// TIA Portal V19 export
FUNCTION "SUBOUTPUT" : Void   // FC4, LAD
{ S7_Optimized_Access := 'TRUE' }
// stored: SetENOAutomatically false
BEGIN

REGION Network 1: HOOTER
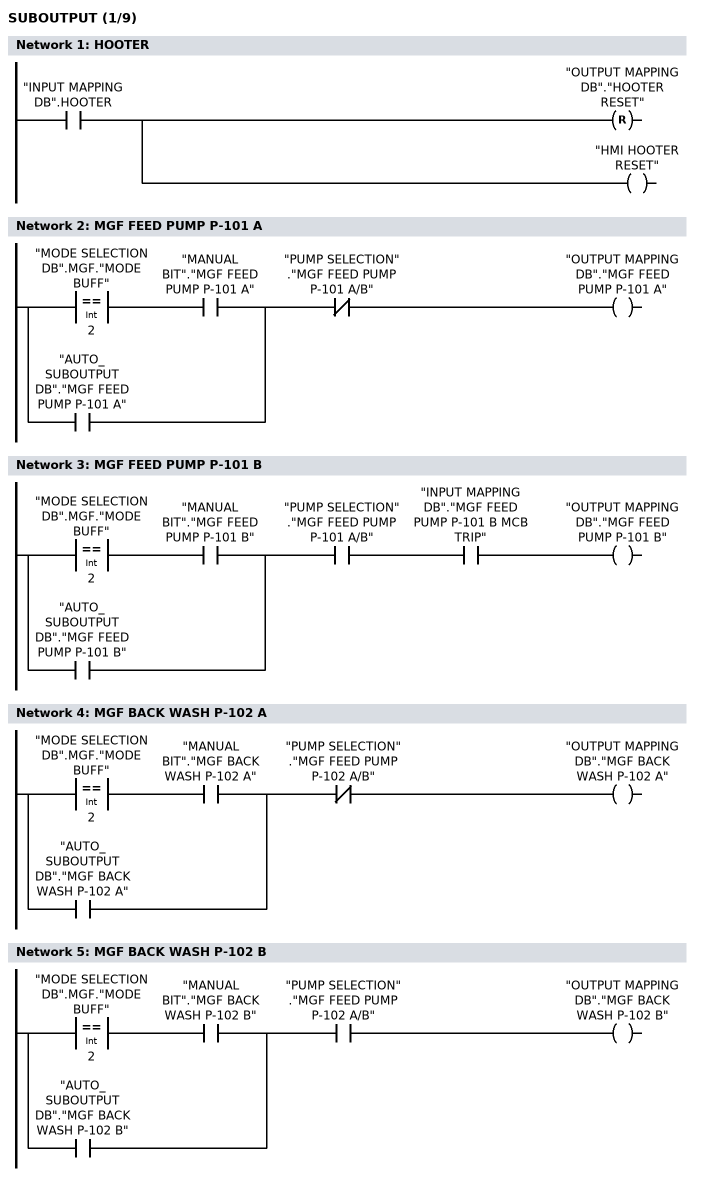
   RUNG wire#powerrail
      Contact( "INPUT MAPPING DB".HOOTER )
      wire#w1
      R_Coil( "OUTPUT MAPPING DB"."HOOTER RESET" )
   END_RUNG
   RUNG wire#w1
      Coil( "HMI HOOTER RESET" )
   END_RUNG
   // the same network as SCL:
   IF "INPUT MAPPING DB".HOOTER THEN "OUTPUT MAPPING DB"."HOOTER RESET" := FALSE; END_IF;
   "HMI HOOTER RESET" := "INPUT MAPPING DB".HOOTER;
END_REGION

REGION Network 2: MGF FEED PUMP P-101 A
   RUNG wire#powerrail
      { S7_Templates := "SrcType := Int" } EQ_Contact(in1 := "MODE SELECTION DB".MGF."MODE BUFF", in2 := 2)
      Contact( "MANUAL BIT"."MGF FEED PUMP P-101 A" )
      wire#w1
      I_Contact( "PUMP SELECTION"."MGF FEED PUMP P-101 A/B" )
      Coil( "OUTPUT MAPPING DB"."MGF FEED PUMP P-101 A" )
   END_RUNG
   RUNG wire#powerrail
      Contact( "AUTO_SUBOUTPUT DB"."MGF FEED PUMP P-101 A" )
   END_RUNG wire#w1
   // the same network as SCL:
   "OUTPUT MAPPING DB"."MGF FEED PUMP P-101 A" := ((("MODE SELECTION DB".MGF."MODE BUFF" = 2) AND "MANUAL BIT"."MGF FEED PUMP P-101 A") OR "AUTO_SUBOUTPUT DB"."MGF FEED PUMP P-101 A") AND NOT "PUMP SELECTION"."MGF FEED PUMP P-101 A/B";
END_REGION

REGION Network 3: MGF FEED PUMP P-101 B
   RUNG wire#powerrail
      { S7_Templates := "SrcType := Int" } EQ_Contact(in1 := "MODE SELECTION DB".MGF."MODE BUFF", in2 := 2)
      Contact( "MANUAL BIT"."MGF FEED PUMP P-101 B" )
      wire#w1
      Contact( "PUMP SELECTION"."MGF FEED PUMP P-101 A/B" )
      Contact( "INPUT MAPPING DB"."MGF FEED PUMP P-101 B MCB TRIP" )
      Coil( "OUTPUT MAPPING DB"."MGF FEED PUMP P-101 B" )
   END_RUNG
   RUNG wire#powerrail
      Contact( "AUTO_SUBOUTPUT DB"."MGF FEED PUMP P-101 B" )
   END_RUNG wire#w1
   // the same network as SCL:
   "OUTPUT MAPPING DB"."MGF FEED PUMP P-101 B" := ((("MODE SELECTION DB".MGF."MODE BUFF" = 2) AND "MANUAL BIT"."MGF FEED PUMP P-101 B") OR "AUTO_SUBOUTPUT DB"."MGF FEED PUMP P-101 B") AND "PUMP SELECTION"."MGF FEED PUMP P-101 A/B" AND "INPUT MAPPING DB"."MGF FEED PUMP P-101 B MCB TRIP";
END_REGION

REGION Network 4: MGF BACK WASH P-102 A
   RUNG wire#powerrail
      { S7_Templates := "SrcType := Int" } EQ_Contact(in1 := "MODE SELECTION DB".MGF."MODE BUFF", in2 := 2)
      Contact( "MANUAL BIT"."MGF BACK WASH P-102 A" )
      wire#w1
      I_Contact( "PUMP SELECTION"."MGF FEED PUMP P-102 A/B" )
      Coil( "OUTPUT MAPPING DB"."MGF BACK WASH P-102 A" )
   END_RUNG
   RUNG wire#powerrail
      Contact( "AUTO_SUBOUTPUT DB"."MGF BACK WASH P-102 A" )
   END_RUNG wire#w1
   // the same network as SCL:
   "OUTPUT MAPPING DB"."MGF BACK WASH P-102 A" := ((("MODE SELECTION DB".MGF."MODE BUFF" = 2) AND "MANUAL BIT"."MGF BACK WASH P-102 A") OR "AUTO_SUBOUTPUT DB"."MGF BACK WASH P-102 A") AND NOT "PUMP SELECTION"."MGF FEED PUMP P-102 A/B";
END_REGION

REGION Network 5: MGF BACK WASH P-102 B
   RUNG wire#powerrail
      { S7_Templates := "SrcType := Int" } EQ_Contact(in1 := "MODE SELECTION DB".MGF."MODE BUFF", in2 := 2)
      Contact( "MANUAL BIT"."MGF BACK WASH P-102 B" )
      wire#w1
      Contact( "PUMP SELECTION"."MGF FEED PUMP P-102 A/B" )
      Coil( "OUTPUT MAPPING DB"."MGF BACK WASH P-102 B" )
   END_RUNG
   RUNG wire#powerrail
      Contact( "AUTO_SUBOUTPUT DB"."MGF BACK WASH P-102 B" )
   END_RUNG wire#w1
   // the same network as SCL:
   "OUTPUT MAPPING DB"."MGF BACK WASH P-102 B" := ((("MODE SELECTION DB".MGF."MODE BUFF" = 2) AND "MANUAL BIT"."MGF BACK WASH P-102 B") OR "AUTO_SUBOUTPUT DB"."MGF BACK WASH P-102 B") AND "PUMP SELECTION"."MGF FEED PUMP P-102 A/B";
END_REGION

REGION Network 6: UF FEED PUMP P-103 A
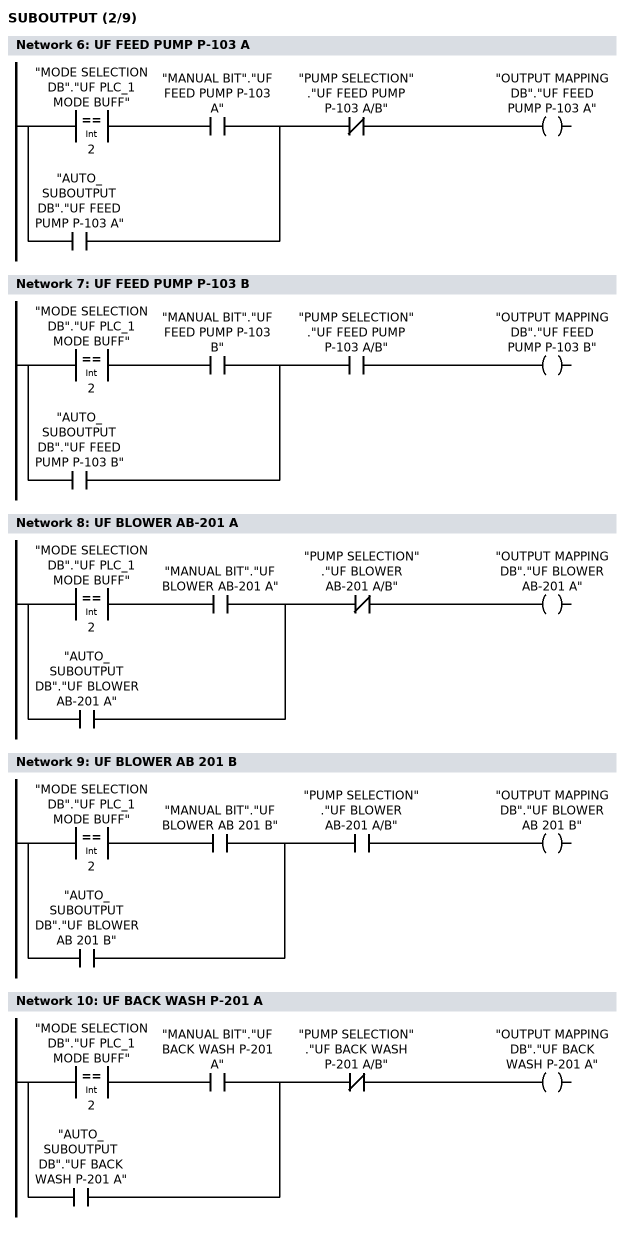
   RUNG wire#powerrail
      { S7_Templates := "SrcType := Int" } EQ_Contact(in1 := "MODE SELECTION DB"."UF PLC_1 MODE BUFF", in2 := 2)
      Contact( "MANUAL BIT"."UF FEED PUMP P-103 A" )
      wire#w1
      I_Contact( "PUMP SELECTION"."UF FEED PUMP P-103 A/B" )
      Coil( "OUTPUT MAPPING DB"."UF FEED PUMP P-103 A" )
   END_RUNG
   RUNG wire#powerrail
      Contact( "AUTO_SUBOUTPUT DB"."UF FEED PUMP P-103 A" )
   END_RUNG wire#w1
   // the same network as SCL:
   "OUTPUT MAPPING DB"."UF FEED PUMP P-103 A" := ((("MODE SELECTION DB"."UF PLC_1 MODE BUFF" = 2) AND "MANUAL BIT"."UF FEED PUMP P-103 A") OR "AUTO_SUBOUTPUT DB"."UF FEED PUMP P-103 A") AND NOT "PUMP SELECTION"."UF FEED PUMP P-103 A/B";
END_REGION

REGION Network 7: UF FEED PUMP P-103 B
   RUNG wire#powerrail
      { S7_Templates := "SrcType := Int" } EQ_Contact(in1 := "MODE SELECTION DB"."UF PLC_1 MODE BUFF", in2 := 2)
      Contact( "MANUAL BIT"."UF FEED PUMP P-103 B" )
      wire#w1
      Contact( "PUMP SELECTION"."UF FEED PUMP P-103 A/B" )
      Coil( "OUTPUT MAPPING DB"."UF FEED PUMP P-103 B" )
   END_RUNG
   RUNG wire#powerrail
      Contact( "AUTO_SUBOUTPUT DB"."UF FEED PUMP P-103 B" )
   END_RUNG wire#w1
   // the same network as SCL:
   "OUTPUT MAPPING DB"."UF FEED PUMP P-103 B" := ((("MODE SELECTION DB"."UF PLC_1 MODE BUFF" = 2) AND "MANUAL BIT"."UF FEED PUMP P-103 B") OR "AUTO_SUBOUTPUT DB"."UF FEED PUMP P-103 B") AND "PUMP SELECTION"."UF FEED PUMP P-103 A/B";
END_REGION

REGION Network 8: UF BLOWER AB-201 A
   RUNG wire#powerrail
      { S7_Templates := "SrcType := Int" } EQ_Contact(in1 := "MODE SELECTION DB"."UF PLC_1 MODE BUFF", in2 := 2)
      Contact( "MANUAL BIT"."UF BLOWER AB-201 A" )
      wire#w1
      I_Contact( "PUMP SELECTION"."UF BLOWER AB-201 A/B" )
      Coil( "OUTPUT MAPPING DB"."UF BLOWER AB-201 A" )
   END_RUNG
   RUNG wire#powerrail
      Contact( "AUTO_SUBOUTPUT DB"."UF BLOWER AB-201 A" )
   END_RUNG wire#w1
   // the same network as SCL:
   "OUTPUT MAPPING DB"."UF BLOWER AB-201 A" := ((("MODE SELECTION DB"."UF PLC_1 MODE BUFF" = 2) AND "MANUAL BIT"."UF BLOWER AB-201 A") OR "AUTO_SUBOUTPUT DB"."UF BLOWER AB-201 A") AND NOT "PUMP SELECTION"."UF BLOWER AB-201 A/B";
END_REGION

REGION Network 9: UF BLOWER AB 201 B
   RUNG wire#powerrail
      { S7_Templates := "SrcType := Int" } EQ_Contact(in1 := "MODE SELECTION DB"."UF PLC_1 MODE BUFF", in2 := 2)
      Contact( "MANUAL BIT"."UF BLOWER AB 201 B" )
      wire#w1
      Contact( "PUMP SELECTION"."UF BLOWER AB-201 A/B" )
      Coil( "OUTPUT MAPPING DB"."UF BLOWER AB 201 B" )
   END_RUNG
   RUNG wire#powerrail
      Contact( "AUTO_SUBOUTPUT DB"."UF BLOWER AB 201 B" )
   END_RUNG wire#w1
   // the same network as SCL:
   "OUTPUT MAPPING DB"."UF BLOWER AB 201 B" := ((("MODE SELECTION DB"."UF PLC_1 MODE BUFF" = 2) AND "MANUAL BIT"."UF BLOWER AB 201 B") OR "AUTO_SUBOUTPUT DB"."UF BLOWER AB 201 B") AND "PUMP SELECTION"."UF BLOWER AB-201 A/B";
END_REGION

REGION Network 10: UF BACK WASH P-201 A
   RUNG wire#powerrail
      { S7_Templates := "SrcType := Int" } EQ_Contact(in1 := "MODE SELECTION DB"."UF PLC_1 MODE BUFF", in2 := 2)
      Contact( "MANUAL BIT"."UF BACK WASH P-201 A" )
      wire#w1
      I_Contact( "PUMP SELECTION"."UF BACK WASH P-201 A/B" )
      Coil( "OUTPUT MAPPING DB"."UF BACK WASH P-201 A" )
   END_RUNG
   RUNG wire#powerrail
      Contact( "AUTO_SUBOUTPUT DB"."UF BACK WASH P-201 A" )
   END_RUNG wire#w1
   // the same network as SCL:
   "OUTPUT MAPPING DB"."UF BACK WASH P-201 A" := ((("MODE SELECTION DB"."UF PLC_1 MODE BUFF" = 2) AND "MANUAL BIT"."UF BACK WASH P-201 A") OR "AUTO_SUBOUTPUT DB"."UF BACK WASH P-201 A") AND NOT "PUMP SELECTION"."UF BACK WASH P-201 A/B";
END_REGION

REGION Network 11: UF BACK WASH P-201 B
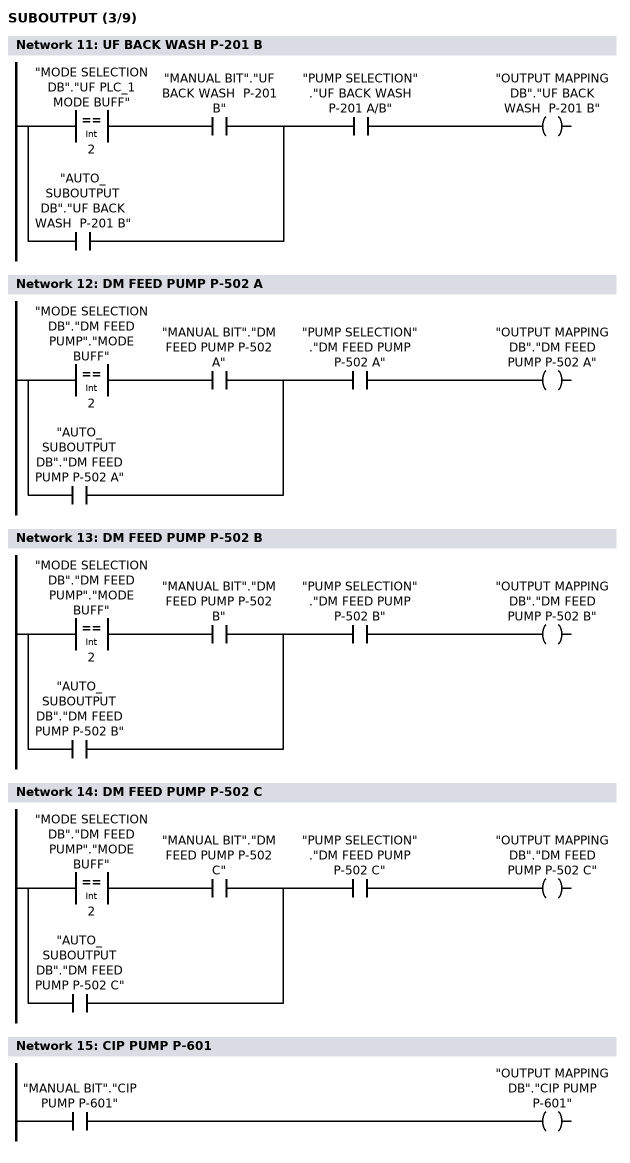
   RUNG wire#powerrail
      { S7_Templates := "SrcType := Int" } EQ_Contact(in1 := "MODE SELECTION DB"."UF PLC_1 MODE BUFF", in2 := 2)
      Contact( "MANUAL BIT"."UF BACK WASH  P-201 B" )
      wire#w1
      Contact( "PUMP SELECTION"."UF BACK WASH P-201 A/B" )
      Coil( "OUTPUT MAPPING DB"."UF BACK WASH  P-201 B" )
   END_RUNG
   RUNG wire#powerrail
      Contact( "AUTO_SUBOUTPUT DB"."UF BACK WASH  P-201 B" )
   END_RUNG wire#w1
   // the same network as SCL:
   "OUTPUT MAPPING DB"."UF BACK WASH  P-201 B" := ((("MODE SELECTION DB"."UF PLC_1 MODE BUFF" = 2) AND "MANUAL BIT"."UF BACK WASH  P-201 B") OR "AUTO_SUBOUTPUT DB"."UF BACK WASH  P-201 B") AND "PUMP SELECTION"."UF BACK WASH P-201 A/B";
END_REGION

REGION Network 12: DM FEED PUMP P-502 A
   RUNG wire#powerrail
      { S7_Templates := "SrcType := Int" } EQ_Contact(in1 := "MODE SELECTION DB"."DM FEED PUMP"."MODE BUFF", in2 := 2)
      Contact( "MANUAL BIT"."DM FEED PUMP P-502 A" )
      wire#w1
      Contact( "PUMP SELECTION"."DM FEED PUMP P-502 A" )
      Coil( "OUTPUT MAPPING DB"."DM FEED PUMP P-502 A" )
   END_RUNG
   RUNG wire#powerrail
      Contact( "AUTO_SUBOUTPUT DB"."DM FEED PUMP P-502 A" )
   END_RUNG wire#w1
   // the same network as SCL:
   "OUTPUT MAPPING DB"."DM FEED PUMP P-502 A" := ((("MODE SELECTION DB"."DM FEED PUMP"."MODE BUFF" = 2) AND "MANUAL BIT"."DM FEED PUMP P-502 A") OR "AUTO_SUBOUTPUT DB"."DM FEED PUMP P-502 A") AND "PUMP SELECTION"."DM FEED PUMP P-502 A";
END_REGION

REGION Network 13: DM FEED PUMP P-502 B
   RUNG wire#powerrail
      { S7_Templates := "SrcType := Int" } EQ_Contact(in1 := "MODE SELECTION DB"."DM FEED PUMP"."MODE BUFF", in2 := 2)
      Contact( "MANUAL BIT"."DM FEED PUMP P-502 B" )
      wire#w1
      Contact( "PUMP SELECTION"."DM FEED PUMP P-502 B" )
      Coil( "OUTPUT MAPPING DB"."DM FEED PUMP P-502 B" )
   END_RUNG
   RUNG wire#powerrail
      Contact( "AUTO_SUBOUTPUT DB"."DM FEED PUMP P-502 B" )
   END_RUNG wire#w1
   // the same network as SCL:
   "OUTPUT MAPPING DB"."DM FEED PUMP P-502 B" := ((("MODE SELECTION DB"."DM FEED PUMP"."MODE BUFF" = 2) AND "MANUAL BIT"."DM FEED PUMP P-502 B") OR "AUTO_SUBOUTPUT DB"."DM FEED PUMP P-502 B") AND "PUMP SELECTION"."DM FEED PUMP P-502 B";
END_REGION

REGION Network 14: DM FEED PUMP P-502 C
   RUNG wire#powerrail
      { S7_Templates := "SrcType := Int" } EQ_Contact(in1 := "MODE SELECTION DB"."DM FEED PUMP"."MODE BUFF", in2 := 2)
      Contact( "MANUAL BIT"."DM FEED PUMP P-502 C" )
      wire#w1
      Contact( "PUMP SELECTION"."DM FEED PUMP P-502 C" )
      Coil( "OUTPUT MAPPING DB"."DM FEED PUMP P-502 C" )
   END_RUNG
   RUNG wire#powerrail
      Contact( "AUTO_SUBOUTPUT DB"."DM FEED PUMP P-502 C" )
   END_RUNG wire#w1
   // the same network as SCL:
   "OUTPUT MAPPING DB"."DM FEED PUMP P-502 C" := ((("MODE SELECTION DB"."DM FEED PUMP"."MODE BUFF" = 2) AND "MANUAL BIT"."DM FEED PUMP P-502 C") OR "AUTO_SUBOUTPUT DB"."DM FEED PUMP P-502 C") AND "PUMP SELECTION"."DM FEED PUMP P-502 C";
END_REGION

REGION Network 15: CIP PUMP P-601
   RUNG wire#powerrail
      Contact( "MANUAL BIT"."CIP PUMP P-601" )
      Coil( "OUTPUT MAPPING DB"."CIP PUMP P-601" )
   END_RUNG
   // the same network as SCL:
   "OUTPUT MAPPING DB"."CIP PUMP P-601" := "MANUAL BIT"."CIP PUMP P-601";
END_REGION

REGION Network 16: BACK WASH RECOVERY P-801 A
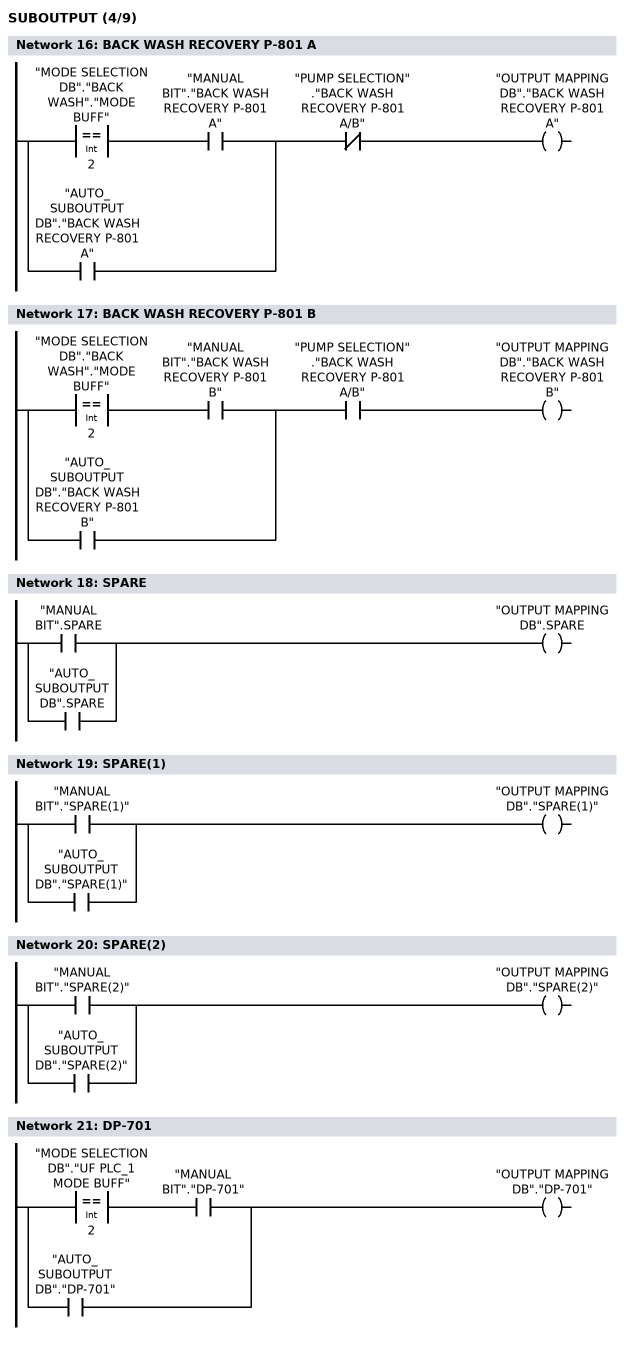
   RUNG wire#powerrail
      { S7_Templates := "SrcType := Int" } EQ_Contact(in1 := "MODE SELECTION DB"."BACK WASH"."MODE BUFF", in2 := 2)
      Contact( "MANUAL BIT"."BACK WASH RECOVERY P-801 A" )
      wire#w1
      I_Contact( "PUMP SELECTION"."BACK WASH RECOVERY P-801 A/B" )
      Coil( "OUTPUT MAPPING DB"."BACK WASH RECOVERY P-801 A" )
   END_RUNG
   RUNG wire#powerrail
      Contact( "AUTO_SUBOUTPUT DB"."BACK WASH RECOVERY P-801 A" )
   END_RUNG wire#w1
   // the same network as SCL:
   "OUTPUT MAPPING DB"."BACK WASH RECOVERY P-801 A" := ((("MODE SELECTION DB"."BACK WASH"."MODE BUFF" = 2) AND "MANUAL BIT"."BACK WASH RECOVERY P-801 A") OR "AUTO_SUBOUTPUT DB"."BACK WASH RECOVERY P-801 A") AND NOT "PUMP SELECTION"."BACK WASH RECOVERY P-801 A/B";
END_REGION

REGION Network 17: BACK WASH RECOVERY P-801 B
   RUNG wire#powerrail
      { S7_Templates := "SrcType := Int" } EQ_Contact(in1 := "MODE SELECTION DB"."BACK WASH"."MODE BUFF", in2 := 2)
      Contact( "MANUAL BIT"."BACK WASH RECOVERY P-801 B" )
      wire#w1
      Contact( "PUMP SELECTION"."BACK WASH RECOVERY P-801 A/B" )
      Coil( "OUTPUT MAPPING DB"."BACK WASH RECOVERY P-801 B" )
   END_RUNG
   RUNG wire#powerrail
      Contact( "AUTO_SUBOUTPUT DB"."BACK WASH RECOVERY P-801 B" )
   END_RUNG wire#w1
   // the same network as SCL:
   "OUTPUT MAPPING DB"."BACK WASH RECOVERY P-801 B" := ((("MODE SELECTION DB"."BACK WASH"."MODE BUFF" = 2) AND "MANUAL BIT"."BACK WASH RECOVERY P-801 B") OR "AUTO_SUBOUTPUT DB"."BACK WASH RECOVERY P-801 B") AND "PUMP SELECTION"."BACK WASH RECOVERY P-801 A/B";
END_REGION

REGION Network 18: SPARE
   RUNG wire#powerrail
      Contact( "MANUAL BIT".SPARE )
      wire#w1
      Coil( "OUTPUT MAPPING DB".SPARE )
   END_RUNG
   RUNG wire#powerrail
      Contact( "AUTO_SUBOUTPUT DB".SPARE )
   END_RUNG wire#w1
   // the same network as SCL:
   "OUTPUT MAPPING DB".SPARE := "MANUAL BIT".SPARE OR "AUTO_SUBOUTPUT DB".SPARE;
END_REGION

REGION Network 19: SPARE(1)
   RUNG wire#powerrail
      Contact( "MANUAL BIT"."SPARE(1)" )
      wire#w1
      Coil( "OUTPUT MAPPING DB"."SPARE(1)" )
   END_RUNG
   RUNG wire#powerrail
      Contact( "AUTO_SUBOUTPUT DB"."SPARE(1)" )
   END_RUNG wire#w1
   // the same network as SCL:
   "OUTPUT MAPPING DB"."SPARE(1)" := "MANUAL BIT"."SPARE(1)" OR "AUTO_SUBOUTPUT DB"."SPARE(1)";
END_REGION

REGION Network 20: SPARE(2)
   RUNG wire#powerrail
      Contact( "MANUAL BIT"."SPARE(2)" )
      wire#w1
      Coil( "OUTPUT MAPPING DB"."SPARE(2)" )
   END_RUNG
   RUNG wire#powerrail
      Contact( "AUTO_SUBOUTPUT DB"."SPARE(2)" )
   END_RUNG wire#w1
   // the same network as SCL:
   "OUTPUT MAPPING DB"."SPARE(2)" := "MANUAL BIT"."SPARE(2)" OR "AUTO_SUBOUTPUT DB"."SPARE(2)";
END_REGION

REGION Network 21: DP-701
   RUNG wire#powerrail
      { S7_Templates := "SrcType := Int" } EQ_Contact(in1 := "MODE SELECTION DB"."UF PLC_1 MODE BUFF", in2 := 2)
      Contact( "MANUAL BIT"."DP-701" )
      wire#w1
      Coil( "OUTPUT MAPPING DB"."DP-701" )
   END_RUNG
   RUNG wire#powerrail
      Contact( "AUTO_SUBOUTPUT DB"."DP-701" )
   END_RUNG wire#w1
   // the same network as SCL:
   "OUTPUT MAPPING DB"."DP-701" := (("MODE SELECTION DB"."UF PLC_1 MODE BUFF" = 2) AND "MANUAL BIT"."DP-701") OR "AUTO_SUBOUTPUT DB"."DP-701";
END_REGION

REGION Network 22: DP-702
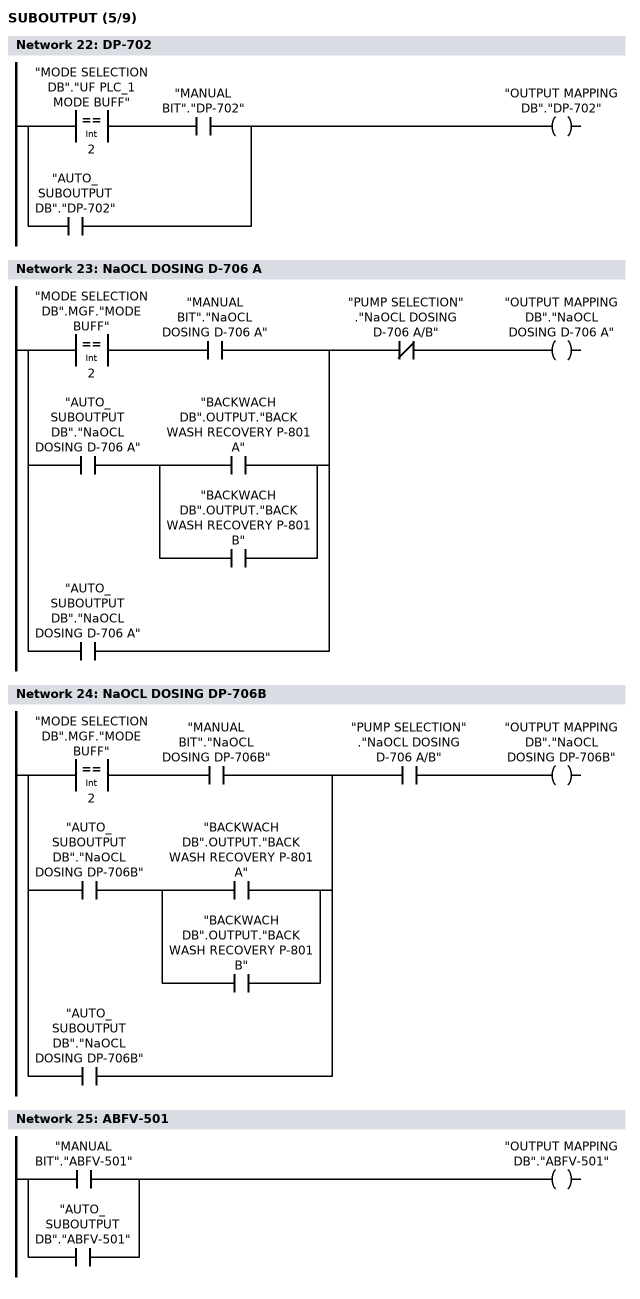
   RUNG wire#powerrail
      { S7_Templates := "SrcType := Int" } EQ_Contact(in1 := "MODE SELECTION DB"."UF PLC_1 MODE BUFF", in2 := 2)
      Contact( "MANUAL BIT"."DP-702" )
      wire#w1
      Coil( "OUTPUT MAPPING DB"."DP-702" )
   END_RUNG
   RUNG wire#powerrail
      Contact( "AUTO_SUBOUTPUT DB"."DP-702" )
   END_RUNG wire#w1
   // the same network as SCL:
   "OUTPUT MAPPING DB"."DP-702" := (("MODE SELECTION DB"."UF PLC_1 MODE BUFF" = 2) AND "MANUAL BIT"."DP-702") OR "AUTO_SUBOUTPUT DB"."DP-702";
END_REGION

REGION Network 23: NaOCL DOSING D-706 A
   RUNG wire#powerrail
      { S7_Templates := "SrcType := Int" } EQ_Contact(in1 := "MODE SELECTION DB".MGF."MODE BUFF", in2 := 2)
      Contact( "MANUAL BIT"."NaOCL DOSING D-706 A" )
      wire#w1
      I_Contact( "PUMP SELECTION"."NaOCL DOSING D-706 A/B" )
      Coil( "OUTPUT MAPPING DB"."NaOCL DOSING D-706 A" )
   END_RUNG
   RUNG wire#powerrail
      Contact( "AUTO_SUBOUTPUT DB"."NaOCL DOSING D-706 A" )
      wire#w2
      Contact( "BACKWACH DB".OUTPUT."BACK WASH RECOVERY P-801 A" )
   END_RUNG wire#w1
   RUNG wire#w2
      Contact( "BACKWACH DB".OUTPUT."BACK WASH RECOVERY P-801 B" )
   END_RUNG wire#w1
   RUNG wire#powerrail
      Contact( "AUTO_SUBOUTPUT DB"."NaOCL DOSING D-706 A" )
   END_RUNG wire#w1
   // the same network as SCL:
   "OUTPUT MAPPING DB"."NaOCL DOSING D-706 A" := ((("MODE SELECTION DB".MGF."MODE BUFF" = 2) AND "MANUAL BIT"."NaOCL DOSING D-706 A") OR ("AUTO_SUBOUTPUT DB"."NaOCL DOSING D-706 A" AND ("BACKWACH DB".OUTPUT."BACK WASH RECOVERY P-801 A" OR "BACKWACH DB".OUTPUT."BACK WASH RECOVERY P-801 B")) OR "AUTO_SUBOUTPUT DB"."NaOCL DOSING D-706 A") AND NOT "PUMP SELECTION"."NaOCL DOSING D-706 A/B";
END_REGION

REGION Network 24: NaOCL DOSING DP-706B
   RUNG wire#powerrail
      { S7_Templates := "SrcType := Int" } EQ_Contact(in1 := "MODE SELECTION DB".MGF."MODE BUFF", in2 := 2)
      Contact( "MANUAL BIT"."NaOCL DOSING DP-706B" )
      wire#w1
      Contact( "PUMP SELECTION"."NaOCL DOSING D-706 A/B" )
      Coil( "OUTPUT MAPPING DB"."NaOCL DOSING DP-706B" )
   END_RUNG
   RUNG wire#powerrail
      Contact( "AUTO_SUBOUTPUT DB"."NaOCL DOSING DP-706B" )
      wire#w2
      Contact( "BACKWACH DB".OUTPUT."BACK WASH RECOVERY P-801 A" )
   END_RUNG wire#w1
   RUNG wire#w2
      Contact( "BACKWACH DB".OUTPUT."BACK WASH RECOVERY P-801 B" )
   END_RUNG wire#w1
   RUNG wire#powerrail
      Contact( "AUTO_SUBOUTPUT DB"."NaOCL DOSING DP-706B" )
   END_RUNG wire#w1
   // the same network as SCL:
   "OUTPUT MAPPING DB"."NaOCL DOSING DP-706B" := ((("MODE SELECTION DB".MGF."MODE BUFF" = 2) AND "MANUAL BIT"."NaOCL DOSING DP-706B") OR ("AUTO_SUBOUTPUT DB"."NaOCL DOSING DP-706B" AND ("BACKWACH DB".OUTPUT."BACK WASH RECOVERY P-801 A" OR "BACKWACH DB".OUTPUT."BACK WASH RECOVERY P-801 B")) OR "AUTO_SUBOUTPUT DB"."NaOCL DOSING DP-706B") AND "PUMP SELECTION"."NaOCL DOSING D-706 A/B";
END_REGION

REGION Network 25: ABFV-501
   RUNG wire#powerrail
      Contact( "MANUAL BIT"."ABFV-501" )
      wire#w1
      Coil( "OUTPUT MAPPING DB"."ABFV-501" )
   END_RUNG
   RUNG wire#powerrail
      Contact( "AUTO_SUBOUTPUT DB"."ABFV-501" )
   END_RUNG wire#w1
   // the same network as SCL:
   "OUTPUT MAPPING DB"."ABFV-501" := "MANUAL BIT"."ABFV-501" OR "AUTO_SUBOUTPUT DB"."ABFV-501";
END_REGION

REGION Network 26: ABFV-502
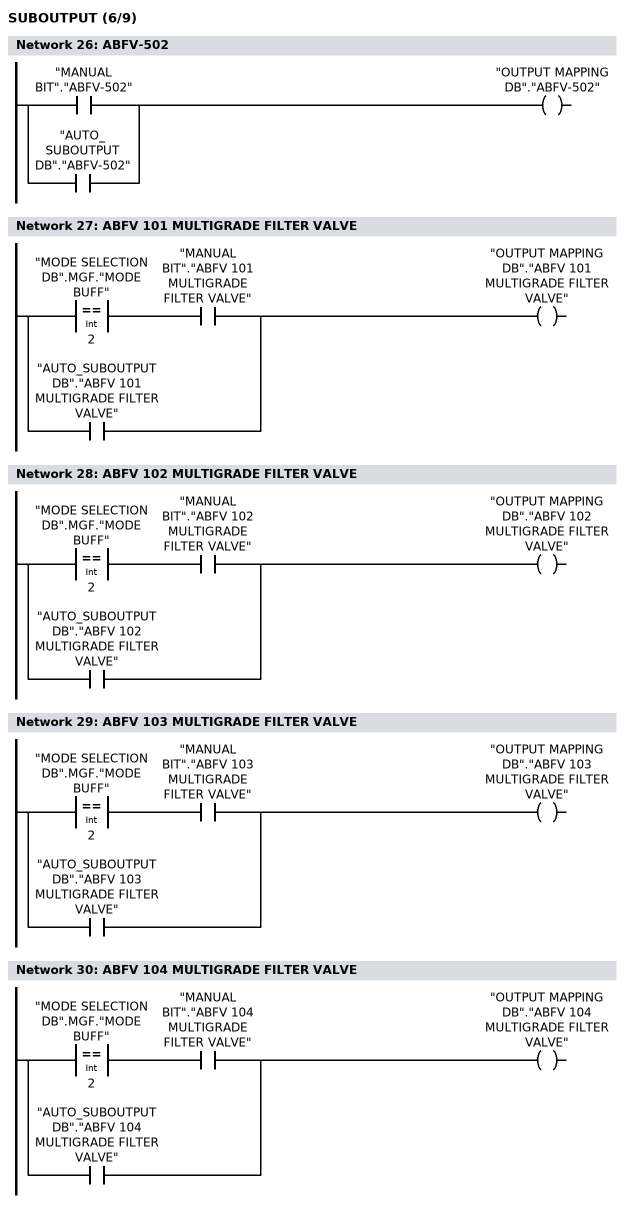
   RUNG wire#powerrail
      Contact( "MANUAL BIT"."ABFV-502" )
      wire#w1
      Coil( "OUTPUT MAPPING DB"."ABFV-502" )
   END_RUNG
   RUNG wire#powerrail
      Contact( "AUTO_SUBOUTPUT DB"."ABFV-502" )
   END_RUNG wire#w1
   // the same network as SCL:
   "OUTPUT MAPPING DB"."ABFV-502" := "MANUAL BIT"."ABFV-502" OR "AUTO_SUBOUTPUT DB"."ABFV-502";
END_REGION

REGION Network 27: ABFV 101 MULTIGRADE FILTER VALVE
   RUNG wire#powerrail
      { S7_Templates := "SrcType := Int" } EQ_Contact(in1 := "MODE SELECTION DB".MGF."MODE BUFF", in2 := 2)
      Contact( "MANUAL BIT"."ABFV 101 MULTIGRADE FILTER VALVE" )
      wire#w1
      Coil( "OUTPUT MAPPING DB"."ABFV 101 MULTIGRADE FILTER VALVE" )
   END_RUNG
   RUNG wire#powerrail
      Contact( "AUTO_SUBOUTPUT DB"."ABFV 101 MULTIGRADE FILTER VALVE" )
   END_RUNG wire#w1
   // the same network as SCL:
   "OUTPUT MAPPING DB"."ABFV 101 MULTIGRADE FILTER VALVE" := (("MODE SELECTION DB".MGF."MODE BUFF" = 2) AND "MANUAL BIT"."ABFV 101 MULTIGRADE FILTER VALVE") OR "AUTO_SUBOUTPUT DB"."ABFV 101 MULTIGRADE FILTER VALVE";
END_REGION

REGION Network 28: ABFV 102 MULTIGRADE FILTER VALVE
   RUNG wire#powerrail
      { S7_Templates := "SrcType := Int" } EQ_Contact(in1 := "MODE SELECTION DB".MGF."MODE BUFF", in2 := 2)
      Contact( "MANUAL BIT"."ABFV 102 MULTIGRADE FILTER VALVE" )
      wire#w1
      Coil( "OUTPUT MAPPING DB"."ABFV 102 MULTIGRADE FILTER VALVE" )
   END_RUNG
   RUNG wire#powerrail
      Contact( "AUTO_SUBOUTPUT DB"."ABFV 102 MULTIGRADE FILTER VALVE" )
   END_RUNG wire#w1
   // the same network as SCL:
   "OUTPUT MAPPING DB"."ABFV 102 MULTIGRADE FILTER VALVE" := (("MODE SELECTION DB".MGF."MODE BUFF" = 2) AND "MANUAL BIT"."ABFV 102 MULTIGRADE FILTER VALVE") OR "AUTO_SUBOUTPUT DB"."ABFV 102 MULTIGRADE FILTER VALVE";
END_REGION

REGION Network 29: ABFV 103 MULTIGRADE FILTER VALVE
   RUNG wire#powerrail
      { S7_Templates := "SrcType := Int" } EQ_Contact(in1 := "MODE SELECTION DB".MGF."MODE BUFF", in2 := 2)
      Contact( "MANUAL BIT"."ABFV 103 MULTIGRADE FILTER VALVE" )
      wire#w1
      Coil( "OUTPUT MAPPING DB"."ABFV 103 MULTIGRADE FILTER VALVE" )
   END_RUNG
   RUNG wire#powerrail
      Contact( "AUTO_SUBOUTPUT DB"."ABFV 103 MULTIGRADE FILTER VALVE" )
   END_RUNG wire#w1
   // the same network as SCL:
   "OUTPUT MAPPING DB"."ABFV 103 MULTIGRADE FILTER VALVE" := (("MODE SELECTION DB".MGF."MODE BUFF" = 2) AND "MANUAL BIT"."ABFV 103 MULTIGRADE FILTER VALVE") OR "AUTO_SUBOUTPUT DB"."ABFV 103 MULTIGRADE FILTER VALVE";
END_REGION

REGION Network 30: ABFV 104 MULTIGRADE FILTER VALVE
   RUNG wire#powerrail
      { S7_Templates := "SrcType := Int" } EQ_Contact(in1 := "MODE SELECTION DB".MGF."MODE BUFF", in2 := 2)
      Contact( "MANUAL BIT"."ABFV 104 MULTIGRADE FILTER VALVE" )
      wire#w1
      Coil( "OUTPUT MAPPING DB"."ABFV 104 MULTIGRADE FILTER VALVE" )
   END_RUNG
   RUNG wire#powerrail
      Contact( "AUTO_SUBOUTPUT DB"."ABFV 104 MULTIGRADE FILTER VALVE" )
   END_RUNG wire#w1
   // the same network as SCL:
   "OUTPUT MAPPING DB"."ABFV 104 MULTIGRADE FILTER VALVE" := (("MODE SELECTION DB".MGF."MODE BUFF" = 2) AND "MANUAL BIT"."ABFV 104 MULTIGRADE FILTER VALVE") OR "AUTO_SUBOUTPUT DB"."ABFV 104 MULTIGRADE FILTER VALVE";
END_REGION

REGION Network 31: ABFV 105 MULTIGRADE FILTER VALVE
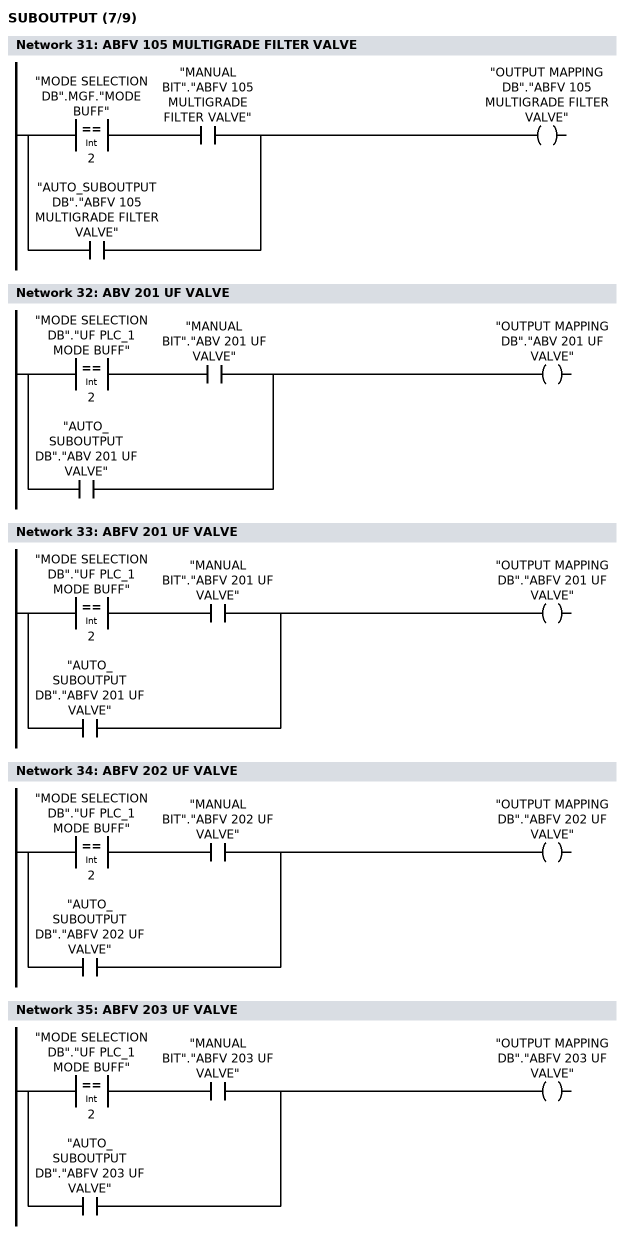
   RUNG wire#powerrail
      { S7_Templates := "SrcType := Int" } EQ_Contact(in1 := "MODE SELECTION DB".MGF."MODE BUFF", in2 := 2)
      Contact( "MANUAL BIT"."ABFV 105 MULTIGRADE FILTER VALVE" )
      wire#w1
      Coil( "OUTPUT MAPPING DB"."ABFV 105 MULTIGRADE FILTER VALVE" )
   END_RUNG
   RUNG wire#powerrail
      Contact( "AUTO_SUBOUTPUT DB"."ABFV 105 MULTIGRADE FILTER VALVE" )
   END_RUNG wire#w1
   // the same network as SCL:
   "OUTPUT MAPPING DB"."ABFV 105 MULTIGRADE FILTER VALVE" := (("MODE SELECTION DB".MGF."MODE BUFF" = 2) AND "MANUAL BIT"."ABFV 105 MULTIGRADE FILTER VALVE") OR "AUTO_SUBOUTPUT DB"."ABFV 105 MULTIGRADE FILTER VALVE";
END_REGION

REGION Network 32: ABV 201 UF VALVE
   RUNG wire#powerrail
      { S7_Templates := "SrcType := Int" } EQ_Contact(in1 := "MODE SELECTION DB"."UF PLC_1 MODE BUFF", in2 := 2)
      Contact( "MANUAL BIT"."ABV 201 UF VALVE" )
      wire#w1
      Coil( "OUTPUT MAPPING DB"."ABV 201 UF VALVE" )
   END_RUNG
   RUNG wire#powerrail
      Contact( "AUTO_SUBOUTPUT DB"."ABV 201 UF VALVE" )
   END_RUNG wire#w1
   // the same network as SCL:
   "OUTPUT MAPPING DB"."ABV 201 UF VALVE" := (("MODE SELECTION DB"."UF PLC_1 MODE BUFF" = 2) AND "MANUAL BIT"."ABV 201 UF VALVE") OR "AUTO_SUBOUTPUT DB"."ABV 201 UF VALVE";
END_REGION

REGION Network 33: ABFV 201 UF VALVE
   RUNG wire#powerrail
      { S7_Templates := "SrcType := Int" } EQ_Contact(in1 := "MODE SELECTION DB"."UF PLC_1 MODE BUFF", in2 := 2)
      Contact( "MANUAL BIT"."ABFV 201 UF VALVE" )
      wire#w1
      Coil( "OUTPUT MAPPING DB"."ABFV 201 UF VALVE" )
   END_RUNG
   RUNG wire#powerrail
      Contact( "AUTO_SUBOUTPUT DB"."ABFV 201 UF VALVE" )
   END_RUNG wire#w1
   // the same network as SCL:
   "OUTPUT MAPPING DB"."ABFV 201 UF VALVE" := (("MODE SELECTION DB"."UF PLC_1 MODE BUFF" = 2) AND "MANUAL BIT"."ABFV 201 UF VALVE") OR "AUTO_SUBOUTPUT DB"."ABFV 201 UF VALVE";
END_REGION

REGION Network 34: ABFV 202 UF VALVE
   RUNG wire#powerrail
      { S7_Templates := "SrcType := Int" } EQ_Contact(in1 := "MODE SELECTION DB"."UF PLC_1 MODE BUFF", in2 := 2)
      Contact( "MANUAL BIT"."ABFV 202 UF VALVE" )
      wire#w1
      Coil( "OUTPUT MAPPING DB"."ABFV 202 UF VALVE" )
   END_RUNG
   RUNG wire#powerrail
      Contact( "AUTO_SUBOUTPUT DB"."ABFV 202 UF VALVE" )
   END_RUNG wire#w1
   // the same network as SCL:
   "OUTPUT MAPPING DB"."ABFV 202 UF VALVE" := (("MODE SELECTION DB"."UF PLC_1 MODE BUFF" = 2) AND "MANUAL BIT"."ABFV 202 UF VALVE") OR "AUTO_SUBOUTPUT DB"."ABFV 202 UF VALVE";
END_REGION

REGION Network 35: ABFV 203 UF VALVE
   RUNG wire#powerrail
      { S7_Templates := "SrcType := Int" } EQ_Contact(in1 := "MODE SELECTION DB"."UF PLC_1 MODE BUFF", in2 := 2)
      Contact( "MANUAL BIT"."ABFV 203 UF VALVE" )
      wire#w1
      Coil( "OUTPUT MAPPING DB"."ABFV 203 UF VALVE" )
   END_RUNG
   RUNG wire#powerrail
      Contact( "AUTO_SUBOUTPUT DB"."ABFV 203 UF VALVE" )
   END_RUNG wire#w1
   // the same network as SCL:
   "OUTPUT MAPPING DB"."ABFV 203 UF VALVE" := (("MODE SELECTION DB"."UF PLC_1 MODE BUFF" = 2) AND "MANUAL BIT"."ABFV 203 UF VALVE") OR "AUTO_SUBOUTPUT DB"."ABFV 203 UF VALVE";
END_REGION

REGION Network 36: ABFV 204 UF VALVE
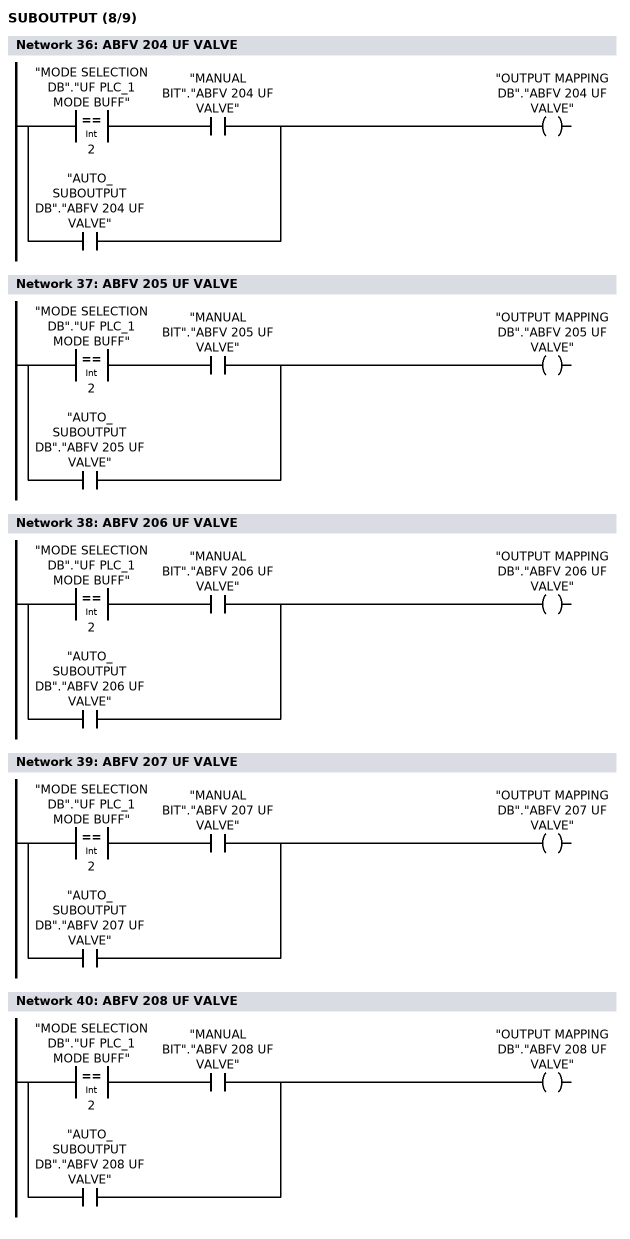
   RUNG wire#powerrail
      { S7_Templates := "SrcType := Int" } EQ_Contact(in1 := "MODE SELECTION DB"."UF PLC_1 MODE BUFF", in2 := 2)
      Contact( "MANUAL BIT"."ABFV 204 UF VALVE" )
      wire#w1
      Coil( "OUTPUT MAPPING DB"."ABFV 204 UF VALVE" )
   END_RUNG
   RUNG wire#powerrail
      Contact( "AUTO_SUBOUTPUT DB"."ABFV 204 UF VALVE" )
   END_RUNG wire#w1
   // the same network as SCL:
   "OUTPUT MAPPING DB"."ABFV 204 UF VALVE" := (("MODE SELECTION DB"."UF PLC_1 MODE BUFF" = 2) AND "MANUAL BIT"."ABFV 204 UF VALVE") OR "AUTO_SUBOUTPUT DB"."ABFV 204 UF VALVE";
END_REGION

REGION Network 37: ABFV 205 UF VALVE
   RUNG wire#powerrail
      { S7_Templates := "SrcType := Int" } EQ_Contact(in1 := "MODE SELECTION DB"."UF PLC_1 MODE BUFF", in2 := 2)
      Contact( "MANUAL BIT"."ABFV 205 UF VALVE" )
      wire#w1
      Coil( "OUTPUT MAPPING DB"."ABFV 205 UF VALVE" )
   END_RUNG
   RUNG wire#powerrail
      Contact( "AUTO_SUBOUTPUT DB"."ABFV 205 UF VALVE" )
   END_RUNG wire#w1
   // the same network as SCL:
   "OUTPUT MAPPING DB"."ABFV 205 UF VALVE" := (("MODE SELECTION DB"."UF PLC_1 MODE BUFF" = 2) AND "MANUAL BIT"."ABFV 205 UF VALVE") OR "AUTO_SUBOUTPUT DB"."ABFV 205 UF VALVE";
END_REGION

REGION Network 38: ABFV 206 UF VALVE
   RUNG wire#powerrail
      { S7_Templates := "SrcType := Int" } EQ_Contact(in1 := "MODE SELECTION DB"."UF PLC_1 MODE BUFF", in2 := 2)
      Contact( "MANUAL BIT"."ABFV 206 UF VALVE" )
      wire#w1
      Coil( "OUTPUT MAPPING DB"."ABFV 206 UF VALVE" )
   END_RUNG
   RUNG wire#powerrail
      Contact( "AUTO_SUBOUTPUT DB"."ABFV 206 UF VALVE" )
   END_RUNG wire#w1
   // the same network as SCL:
   "OUTPUT MAPPING DB"."ABFV 206 UF VALVE" := (("MODE SELECTION DB"."UF PLC_1 MODE BUFF" = 2) AND "MANUAL BIT"."ABFV 206 UF VALVE") OR "AUTO_SUBOUTPUT DB"."ABFV 206 UF VALVE";
END_REGION

REGION Network 39: ABFV 207 UF VALVE
   RUNG wire#powerrail
      { S7_Templates := "SrcType := Int" } EQ_Contact(in1 := "MODE SELECTION DB"."UF PLC_1 MODE BUFF", in2 := 2)
      Contact( "MANUAL BIT"."ABFV 207 UF VALVE" )
      wire#w1
      Coil( "OUTPUT MAPPING DB"."ABFV 207 UF VALVE" )
   END_RUNG
   RUNG wire#powerrail
      Contact( "AUTO_SUBOUTPUT DB"."ABFV 207 UF VALVE" )
   END_RUNG wire#w1
   // the same network as SCL:
   "OUTPUT MAPPING DB"."ABFV 207 UF VALVE" := (("MODE SELECTION DB"."UF PLC_1 MODE BUFF" = 2) AND "MANUAL BIT"."ABFV 207 UF VALVE") OR "AUTO_SUBOUTPUT DB"."ABFV 207 UF VALVE";
END_REGION

REGION Network 40: ABFV 208 UF VALVE
   RUNG wire#powerrail
      { S7_Templates := "SrcType := Int" } EQ_Contact(in1 := "MODE SELECTION DB"."UF PLC_1 MODE BUFF", in2 := 2)
      Contact( "MANUAL BIT"."ABFV 208 UF VALVE" )
      wire#w1
      Coil( "OUTPUT MAPPING DB"."ABFV 208 UF VALVE" )
   END_RUNG
   RUNG wire#powerrail
      Contact( "AUTO_SUBOUTPUT DB"."ABFV 208 UF VALVE" )
   END_RUNG wire#w1
   // the same network as SCL:
   "OUTPUT MAPPING DB"."ABFV 208 UF VALVE" := (("MODE SELECTION DB"."UF PLC_1 MODE BUFF" = 2) AND "MANUAL BIT"."ABFV 208 UF VALVE") OR "AUTO_SUBOUTPUT DB"."ABFV 208 UF VALVE";
END_REGION

REGION Network 41: UV 601
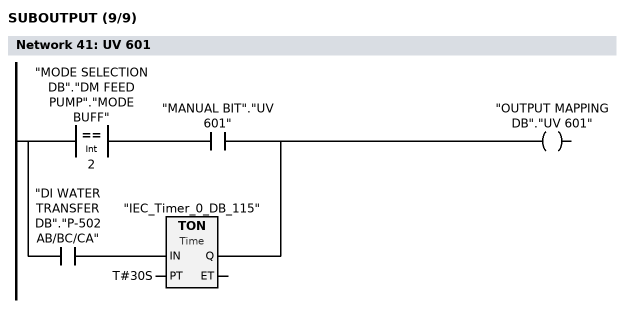
   RUNG wire#powerrail
      { S7_Templates := "SrcType := Int" } EQ_Contact(in1 := "MODE SELECTION DB"."DM FEED PUMP"."MODE BUFF", in2 := 2)
      Contact( "MANUAL BIT"."UV 601" )
      wire#w1
      Coil( "OUTPUT MAPPING DB"."UV 601" )
   END_RUNG
   RUNG wire#powerrail
      Contact( "DI WATER TRANSFER DB"."P-502 AB/BC/CA" )
      { S7_Templates := "time_type := Time" } "IEC_Timer_0_DB_115".TON(pt := T#30S, et =>)
   END_RUNG wire#w1
   // the same network as SCL:
   "IEC_Timer_0_DB_115".TON(IN := "DI WATER TRANSFER DB"."P-502 AB/BC/CA", PT := T#30S);
   "OUTPUT MAPPING DB"."UV 601" := (("MODE SELECTION DB"."DM FEED PUMP"."MODE BUFF" = 2) AND "MANUAL BIT"."UV 601") OR "IEC_Timer_0_DB_115".Q;
END_REGION
END_FUNCTION
